Staubli VAL3: clkValve15.pgx

program clkValve15()
begin
  call toggleValve(15)
end
